PROGRAM MAIN
VAR
END_VAR

END_PROGRAM

(* stored: Version 1.1.0.1
   POU MAIN: Id {81899879-92e4-47e3-94c8-cb78581e6884}, SpecialFunc None *)
